// TIA Portal V17 export
// export: Created 2024-08-26T21:07:21.3248901Z, ExportSetting WithDefaults, DisplayName Totally Integrated Automation Portal, DisplayVersion V17 Update 7, DisplayName TIA Portal Openness, DisplayVersion V17 Update 7, DisplayName TIA Portal Version Control Interface, DisplayVersion V17, DisplayName SINAMICS Startdrive Advanced, DisplayVersion V17 SP2, DisplayName SINAMICS Startdrive G110M, G120, G120C, G120D, G120P, G115D, DisplayVersion V17 SP2, DisplayName SINAMICS Startdrive G130, G150, S120, S150, SINAMICS MV, S210, DisplayVersion V17 SP2, DisplayName STEP 7 Professional, DisplayVersion V17 Update 7, DisplayName STEP 7 Safety, DisplayVersion V17 Update 6, DisplayName WinCC Advanced / Unified PC, DisplayVersion V17 Update 7
VAR_GLOBAL   // PLC tag table "Default tag table"
   optoSignal AT %I0.7 : Bool;
   nestScannerBusy AT %I3.0 : Bool;
   nestScannerComplete AT %I4.0 : Bool;
   nestScannerError AT %I5.0 : Bool;
   nestScannerDataSize AT %IW334 : Int;
   upperScannerReading AT %I9.0 : Bool;
   upperScannerReadingComplete AT %I10.0 : Bool;
   upperScannerError AT %I11.0 : Bool;
   upperScannerDataSize AT %IW470 : Int;
   angleScannerDataSize AT %IW385 : Int;
   angleScannerBusy AT %I39.0 : Bool;
   angleScannerReadingComplete AT %I40.0 : Bool;
   angleScannerError AT %I41.0 : Bool;
   amgeScannerDataSize AT %IW606 : Int;
   Tag_1 AT %I46.3 : Bool;
   Tag_2 AT %I46.4 : Bool;
   washerPresence AT %I1.0 : Bool;
   toolingID2 AT %I1.6 : Bool;
   finalTorqueAngle AT %IW17 : Word;
   OutputPin2 AT %QB147 : Byte;
   byte0 AT %QB156 : Byte;
   runlight AT %Q159.2 : Bool;
   byte6 AT %QB162 : Byte;
   byte2 AT %QB158 : Byte;
   byte7 AT %QB163 : Byte;
   segmentLight AT %Q159.0 : Bool;
   byte1 AT %QB157 : Byte;
   byte4 AT %QB160 : Byte;
   byte3 AT %QB159 : Byte;
   byte5 AT %QB161 : Byte;
   optoGreen AT %Q1.2 : Bool;
   optoRed AT %Q1.3 : Bool;
   optoYellow AT %Q1.4 : Bool;
   qYellowTurretBlinking AT %Q2.1 : Bool;
   nestScannerRequest AT %Q3.0 : Bool;
   clearUpperScannerReadComplete AT %Q9.0 : Bool;
   upperScannerRequest AT %Q8.0 : Bool;
   angleScannerRequest AT %Q13.0 : Bool;
   clearAngleScannerComplete AT %Q14.0 : Bool;
   clearTorque AT %Q17.5 : Bool;
   System_Byte AT %MB0 : Byte;
   DiagStatusUpdate AT %M0.1 : Bool;
   "CONFIG INICIAL" AT %M89.5 : Bool;
   "CONFIG CILINDROS ON" AT %M89.7 : Bool;
END_VAR
VAR_GLOBAL CONSTANT   // user constants
   "MODELO MOTOR 1" : String := '592';
   "MODELO MOTOR 2" : String := '202';
   "MODELO MOTOR 3" : String := '277';
   "MODELO MOTOR 4" : String := '984';
   "MODELO TRACK L 1" : String := '610';
   "MODELO TRACK L 2" : String := '618';
   "MODELO TRACK L 3" : String := '333';
   "MODELO TRACK L 4" : String := '444';
   "MODELO TRACK L 5" : String := '555';
   "MODELO TRACK L 6" : String := '666';
   "MODELO TRACK L 7" : String := '777';
   "MODELO TRACK L 8" : String := '888';
   "MODELO TRACK R 1" : String := '612';
   "MODELO TRACK R 2" : String := '623';
   "MODELO TRACK R 3" : String := '993';
   "MODELO TRACK R 4" : String := '994';
   "MODELO TRACK R 5" : String := '995';
   "MODELO TRACK R 6" : String := '996';
   "MODELO TRACK R 7" : String := '997';
   "MODELO TRACK R 8" : String := '998';
END_VAR
